# EPICS substitutions: support/adas/iocBoot/iocAdas/boot/icv196.substitutions
#******************************************************************************
# C.E.A. - JWST/MIRI project
#
# "@(#) $Id: icv196.substitutions 23 2013-03-13 15:38:34Z lussi $"
#
# who       when      what
# --------  --------  ----------------------------------------------
# ylussign  26/10/07  created
#
#******************************************************************************
#

file "$(ADAS)/db/BI.template"
{
pattern { DV     , C , S  , P          , SC         , EV }
        { ICV196 , 0 ,  0 , "event 10" , "1 second" , 10 }
        { ICV196 , 0 ,  1 , "event 11" , "1 second" , 11 }
        { ICV196 , 0 ,  2 , ""         , "Event"    , 10 }
        { ICV196 , 0 ,  3 , ""         , "Event"    , 11 }
        { ICV196 , 0 ,  8 , ""         , "1 second" , 0 }
        { ICV196 , 0 ,  9 , ""         , "1 second" , 0 }
        { ICV196 , 0 , 10 , ""         , "1 second" , 0 }
        { ICV196 , 0 , 11 , ""         , "1 second" , 0 }
}

file "$(ADAS)/db/BO.template"
{
pattern { DV     , C , S  }
        { ICV196 , 0 , 16 }
        { ICV196 , 0 , 17 }
        { ICV196 , 0 , 18 }
        { ICV196 , 0 , 19 }
}

file "$(ADAS)/db/MBBI.template"
{
pattern { DV     , C , S  , NB , SC         , EV }
        { ICV196 , 0 , 24 ,  2 , "1 second" , 0 }
        { ICV196 , 0 , 26 ,  6 , "1 second" , 0 }
        { ICV196 , 0 , 44 , 12 , "1 second" , 0 }
        { ICV196 , 0 , 64 ,  8 , "1 second" , 0 }
        { ICV196 , 0 , 88 ,  8 , "1 second" , 0 }
}

file "$(ADAS)/db/MBBO.template"
{
pattern { DV     , C , S  , NB }
        { ICV196 , 0 , 20 ,  4 }
        { ICV196 , 0 , 32 ,  6 }
        { ICV196 , 0 , 56 ,  8 }
        { ICV196 , 0 , 72 , 16 }
}

file "$(ADAS)/db/MBBIDIRECT.template"
{
pattern { DV     , C , S  , NB , SC         , EV }
        { ICV196 , 0 , 24 ,  2 , "1 second" , 0 }
        { ICV196 , 0 , 26 ,  6 , "1 second" , 0 }
}

file "$(ADAS)/db/MBBODIRECT.template"
{
pattern { DV     , C , S  , NB }
        { ICV196 , 0 , 38 ,  2 }
}
